// TIA Portal V19 export
FUNCTION "Trapezoidal_RampTime_1" : LReal   // FC163, LAD
// stored: SetENOAutomatically false
   VAR_INPUT
      VDelta : LReal;   // Delta Final - Initial velocity (mm/min)
      AccDec : LReal;   // Acceleration or Deceleration (mm/s^2)
      Jerk : LReal;   // Jerk (mm/S^3)
   END_VAR
   VAR_TEMP
      VDelta_mm_s : LReal;
      TimeRamp : LReal;
      TimeSmooth : LReal;
      TimeTot : LReal;
   END_VAR
   // Ret_Val : seconds
BEGIN

REGION Network 1 (SCL): seconds
   #Trapezoidal_RampTime_1 := 0.0;


   IF ABS(#VDelta) = 0.0 OR #AccDec <= 0.0 THEN
       RETURN;
   END_IF;


   #VDelta_mm_s := ABS(#VDelta / 60.0);

   #TimeRamp := #VDelta_mm_s / #AccDec;


   IF #TimeRamp > 0.0 AND #Jerk > 0.0 THEN
       #TimeSmooth := #AccDec / #Jerk;
   ELSE
       #TimeSmooth := 0.0;
   END_IF;

   #Trapezoidal_RampTime_1 := #TimeRamp + #TimeSmooth;
END_REGION
END_FUNCTION
